FUNCTION_BLOCK fb_auto
VAR_INPUT
END_VAR
VAR_OUTPUT
END_VAR
VAR
	SFCInit: BOOL;
	trn_paramInitDone: BOOL;
	trn_moveToHomeDone: BOOL;
	trn_removeLensDone: BOOL;
	fbi_paramInit: fb_paramInit;
	var_process: INT;
	flg_tranHomeDone: BOOL;
	flg_sampleHomeDone: BOOL;
	flg_trayHomeDone: BOOL;
	flg_chuckHomeDone: BOOL;
	flg_axisHomeDone: BOOL;
	fbi_lensTranport: fb_lensTranport;
	fbi_palletizeing: fb_palletizeing;
	fbi_gm_measurementModule: fb_gm_measurementModule;
	fbi_gm_transport: fb_gm_transport;
	flg_pushHomeDone: BOOL;
	flg_rotaryHomeDone: BOOL;
	trn_measurementSystemHomeDone: BOOL;
	fbi_debuger : fb_debuger;
	fbi_gateLengthList: fb_gateLengthList;
	fbi_dataSampling: fb_dataSampling;
	timer: TON;
	timer2: TON;
	fbi_gm_removeLens: fb_gm_removeLens;
END_VAR

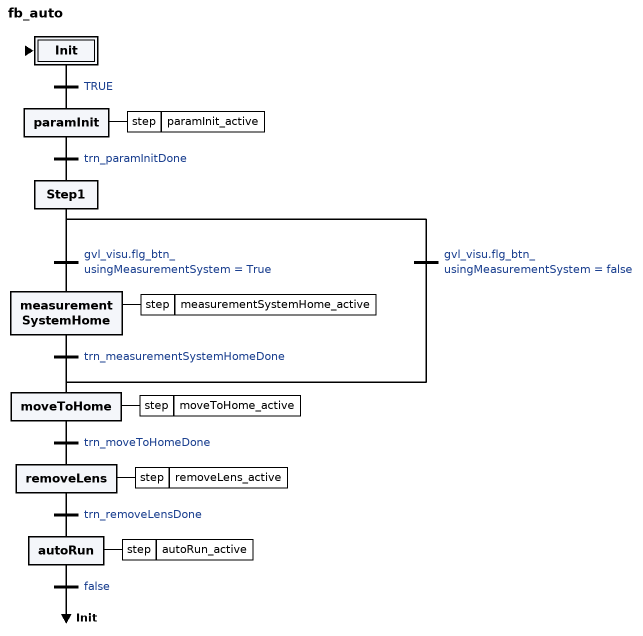
INITIAL_STEP Init:
END_STEP
TRANSITION FROM Init TO paramInit
    := TRUE;
END_TRANSITION
STEP paramInit:
    paramInit_active(N);  // step action
END_STEP
TRANSITION FROM paramInit TO Step1
    := trn_paramInitDone;
END_TRANSITION
STEP Step1:
END_STEP
TRANSITION FROM Step1 TO measurementSystemHome
    := gvl_visu.flg_btn_usingMeasurementSystem = True;
END_TRANSITION
STEP measurementSystemHome:
    measurementSystemHome_active(N);  // step action
END_STEP
TRANSITION FROM measurementSystemHome TO moveToHome
    := trn_measurementSystemHomeDone;
END_TRANSITION
TRANSITION FROM Step1 TO moveToHome
    := gvl_visu.flg_btn_usingMeasurementSystem = false;
END_TRANSITION
STEP moveToHome:
    moveToHome_active(N);  // step action
END_STEP
TRANSITION FROM moveToHome TO removeLens
    := trn_moveToHomeDone;
END_TRANSITION
STEP removeLens:
    removeLens_active(N);  // step action
END_STEP
TRANSITION FROM removeLens TO autoRun
    := trn_removeLensDone;
END_TRANSITION
STEP autoRun:
    autoRun_active(N);  // step action
END_STEP
TRANSITION FROM autoRun TO Init
    := false;
END_TRANSITION

ACTION autoRun_active:
IF autoRun._x AND autoRun.x = FALSE THEN
	THIS^.fbi_lensTranport();
	THIS^.fbi_lensTranport.p_Init := TRUE;
	THIS^.fbi_palletizeing();
	THIS^.fbi_palletizeing.p_Init := TRUE;
	THIS^.fbi_gm_measurementModule.SFCInit := TRUE;
	THIS^.fbi_gm_measurementModule();
	THIS^.fbi_gm_transport();
	THIS^.fbi_gm_transport.p_Init := TRUE;
ELSIF autoRun._x AND autoRun.x THEN
	THIS^.fbi_lensTranport();
	THIS^.fbi_lensTranport.p_Init := FALSE;
	THIS^.fbi_palletizeing();
	THIS^.fbi_palletizeing.p_Init := FALSE;
	IF gvl_visu.flg_btn_usingMeasurementSystem THEN
		THIS^.fbi_gm_measurementModule();
		THIS^.fbi_gm_measurementModule.SFCInit := FALSE;
		THIS^.fbi_gm_transport();
		THIS^.fbi_gm_transport.p_Init := FALSE;
	END_IF
	fbi_dataSampling(
	in_flg_run:= gvl_auto.flg_dataSampling_run, 
	in_var_cavNo:= gvl_auto.buf_cavNo, 
	in_var_pocketNo:= gvl_auto.pocketNo[gvl_auto.buf_cavNo], 
	in_var_gateLength:= gvl_auto.buf_gateLength, 
	in_var_date:= gvl_visu.var_DT, 
	in_flg_nonDefective:= gvl_auto.flg_DataSample_nonDefective, 
	in_flg_defective:= gvl_auto.flg_DataSample_defective, 
	in_flg_sample:= gvl_auto.flg_DataSamle_sample, 
	in_flg_reset:= , 
	ref_dataSet:= gvl_auto.var_DataSet);

	fbi_gateLengthList();
	
	fbi_debuger(
	in_flg_run:= gvl_debug.flg_debug_run, 
	in_flg_start:= gvl_debug.flg_debug_run, 
	in_var_cavQty:= gvl_param.var_productInfo[gvl_param.var_currentProductID].cavQty, 
	out_flg_gateLengthISSuccessed=> gvl_debug.flg_passingMeasurement, 
	out_flg_dummySignal=> , 
	out_flg_lensSetDone=> gvl_debug.out_lensSetDone, 
	out_flg_fiberSens=> gvl_debug.out_fiberSens, 
	out_flg_busy=> gvl_debug.out_busy, 
	out_cav=> gvl_debug.var_cav);
	
END_IF
END_ACTION

ACTION measurementSystemHome_active:
IF measurementSystemHome._x AND measurementSystemHome.x = FALSE THEN
	trn_measurementSystemHomeDone := FALSE;
	gvl_auto.gm_rotaryPowerOn := FALSE;
	var_process := 0;
ELSIF measurementSystemHome._x AND measurementSystemHome.x THEN
	IF gvl_visu.flg_btn_usingMeasurementSystem THEN
		CASE var_process OF
			0://insert parameter
				gvl_solv.fbi_gm_ejector.in_flg_run := FALSE;
				gvl_solv.fbi_gm_chuck.in_flg_run := FALSE;
				gvl_solv.fbi_gm_push.in_flg_run := FALSE;
				gvl_solv.fbi_gm_pickup.in_flg_run := FALSE;
				gvl_solv.fbi_gm_rotary.in_flg_run := FALSE;
				gvl_solv.fbi_gm_stamp.in_flg_run := FALSE;
				gvl_elecylinder.fbi_gm_axisPickUp.in_flg_run := FALSE;
				gvl_elecylinder.fbi_gm_axisTransport.in_flg_run := FALSE;
				gvl_solv.fbi_gm_ejector.in_var_vacMode := eP_ejeVacMode.halt;
				gvl_solv.fbi_gm_chuck.in_var_moveMode := eP_svMoveMode.svA;
				gvl_solv.fbi_gm_push.in_var_moveMode := eP_svMoveMode.svA;
				gvl_solv.fbi_gm_pickup.in_var_moveMode := eP_svMoveMode.svA;
				gvl_solv.fbi_gm_rotary.in_var_moveMode := eP_svMoveMode.svA;
				gvl_solv.fbi_gm_stamp.in_var_moveMode := eP_svMoveMode.svA;
				gvl_elecylinder.fbi_gm_axisPickUp.in_var_moveMode := eP_eleMoveMode.eleA;
				gvl_elecylinder.fbi_gm_axisTransport.in_var_moveMode := eP_eleMoveMode.eleA;
				gvl_axis.ref_r.Position := gvl_param.var_productInfo[gvl_param.var_currentProductID].teachPos.gm_rotary.origin;
				gvl_auto.gm_rotaryPowerOn := TRUE;
				IF gvl_axis.fbi_mc_powerR.Status THEN
					var_process := 1;
				END_IF
			1://first move
				gvl_solv.fbi_gm_ejector.in_flg_run := TRUE;
				gvl_solv.fbi_gm_chuck.in_flg_run := TRUE;
				gvl_solv.fbi_gm_push.in_flg_run := TRUE;
				gvl_elecylinder.fbi_gm_axisPickUp.in_flg_run := TRUE;
				gvl_elecylinder.fbi_gm_axisTransport.in_flg_run := TRUE;
				IF gvl_solv.ref_gm_chuck.in.in_flg_sensA AND
				   gvl_solv.ref_gm_push.in.in_flg_sensA AND
				   gvl_elecylinder.ref_gm_axisPickUp.input.in_flg_sensA AND 
				   gvl_elecylinder.ref_gm_axisTransport.input.in_flg_sensA THEN
				   	gvl_solv.fbi_gm_ejector.in_flg_run := FALSE;
					gvl_solv.fbi_gm_chuck.in_flg_run := FALSE;
					gvl_solv.fbi_gm_push.in_flg_run := FALSE;
					gvl_elecylinder.fbi_gm_axisPickUp .in_flg_run := FALSE;
					gvl_elecylinder.fbi_gm_axisTransport.in_flg_run := FALSE;
					var_process := 2;
				END_IF
			2://second move	
				gvl_axis.ref_r.Execute := TRUE;
				IF gvl_axis.ref_r.Done THEN
					gvl_axis.ref_r.Execute := FALSE;
					var_process := 3;
				END_IF
			3://third move
				gvl_solv.fbi_gm_pickup.in_flg_run := TRUE;
				gvl_solv.fbi_gm_rotary.in_flg_run := TRUE;
				gvl_solv.fbi_gm_stamp.in_flg_run := TRUE;
				IF gvl_solv.ref_gm_pickUp.in.in_flg_sensA AND gvl_solv.ref_gm_rotary.in.in_flg_sensA AND gvl_solv.ref_gm_stamp.in.in_flg_sensA THEN
					var_process := 4;
				END_IF
			4:	
				trn_measurementSystemHomeDone := TRUE;
		END_CASE
		IF gvl_axis.ref_r.Error THEN
			gvl_axis.ref_r.Execute := false;
			var_process := 100;
		END_IF
	ELSE
		trn_measurementSystemHomeDone := TRUE;
	END_IF
END_IF
END_ACTION

ACTION moveToHome_active:
IF moveToHome._x AND moveToHome.x = FALSE THEN
	var_process := 0;
	trn_moveToHomeDone := FALSE;
	gvl_auto.motorPowerOn := FALSE;
ELSIF moveToHome._x AND moveToHome.x THEN
	CASE var_process OF
		0:
			gvl_auto.motorPowerOn := TRUE;
			IF gvl_axis.flg_motorReady THEN
				var_process := 1;
			END_IF
		1://move axisZ
			gvl_axis.ref_z.Position := 0;
			gvl_axis.ref_z.Execute := TRUE;
			IF gvl_axis.ref_z.Done THEN
				gvl_axis.ref_z.Execute := FALSE;
				var_process := 2;
			END_IF
		2://insert parameter
			gvl_solv.fbi_push.in_flg_run := FALSE;
			gvl_elecylinder.fbi_axisTransport.in_var_moveMode := eP_eleMoveMode.eleA;
			gvl_elecylinder.fbi_axisSample.in_var_moveMode := eP_eleMoveMode.eleA;
			gvl_elecylinder.fbi_axisRotary.in_var_moveMode := eP_eleMoveMode.eleA;
			gvl_solv.fbi_chuck.in_var_moveMode := eP_svMoveMode.svA;
			gvl_solv.fbi_push.in_var_moveMode := eP_svMoveMode.svA;
			gvl_elecylinder.fbi_axisTransport.in_flg_run := FALSE;
			gvl_elecylinder.fbi_axisSample.in_flg_run := FALSE;
			gvl_elecylinder.fbi_axisRotary.in_flg_run := FALSE;
			gvl_solv.fbi_chuck.in_flg_run := FALSE;
			gvl_solv.fbi_push.in_flg_run := FALSE;
			gvl_axis.fbi_motionControler.in_flg_start := false;
			gvl_axis.fbi_motionControler.in_var_targetPosX := gvl_param.var_productInfo[gvl_param.var_currentProductID].teachPos.initial.x;
			gvl_axis.fbi_motionControler.in_var_targetPosY := gvl_param.var_productInfo[gvl_param.var_currentProductID].teachPos.initial.y;
			gvl_axis.fbi_motionControler.in_var_targetPosZ := gvl_param.var_productInfo[gvl_param.var_currentProductID].teachPos.initial.z;
			gvl_axis.fbi_motionControler.in_var_direction := eP_motionDirection.XYZ;
			var_process := 3;
		3://moving start
			gvl_elecylinder.fbi_axisTransport.in_flg_run := TRUE;
			gvl_elecylinder.fbi_axisSample.in_flg_run := TRUE;
			gvl_elecylinder.fbi_axisRotary.in_flg_run := TRUE;
			gvl_solv.fbi_chuck.in_flg_run := TRUE;
			gvl_solv.fbi_push.in_flg_run := TRUE;
			gvl_axis.fbi_motionControler.in_flg_start := TRUE;
			IF gvl_elecylinder.fbi_axisTransport.out_flg_Done THEN
				flg_tranHomeDone := TRUE;
			END_IF
			IF gvl_elecylinder.fbi_axisSample.out_flg_Done THEN
				flg_sampleHomeDone := TRUE;
			END_IF
			IF gvl_elecylinder.fbi_axisRotary.out_flg_Done THEN
				flg_rotaryHomeDone := TRUE;
			END_IF
			IF gvl_solv.fbi_chuck.out_flg_Done THEN
				flg_chuckHomeDone := TRUE;
			END_IF
			IF gvl_solv.fbi_push.out_flg_Done THEN
				flg_pushHomeDone := TRUE;
			END_IF
			IF gvl_axis.fbi_motionControler.out_flg_Done THEN
				flg_axisHomeDone := TRUE;
			END_IF 
			IF flg_tranHomeDone AND flg_sampleHomeDone AND flg_chuckHomeDone AND flg_axisHomeDone AND flg_pushHomeDone AND flg_rotaryHomeDone THEN
				var_process := 4;
			END_IF
		4://clear flag
			flg_tranHomeDone := FALSE;
			flg_sampleHomeDone := FALSE;
			flg_chuckHomeDone := FALSE;
			flg_pushHomeDone := FALSE;
			flg_axisHomeDone := FALSE;
			flg_rotaryHomeDone := FALSE;
			gvl_elecylinder.fbi_axisTransport.in_flg_run := FALSE;
			gvl_elecylinder.fbi_axisSample.in_flg_run := FALSE;
			gvl_elecylinder.fbi_axisTrayChange.in_flg_run := FALSE;
			gvl_elecylinder.fbi_axisRotary.in_flg_run := FALSE;
			gvl_solv.fbi_chuck.in_flg_run := FALSE;
			gvl_solv.fbi_push.in_flg_run := FALSE;
			gvl_axis.fbi_motionControler.in_flg_start := FALSE;
			var_process := 5;
		5://check position
			trn_moveToHomeDone := TRUE;			
	END_CASE
END_IF
END_ACTION

PROPERTY p_Init : BOOL
GET
p_Init := THIS^.SFCInit;
END_GET
SET
THIS^.SFCInit := p_Init;
END_SET
END_PROPERTY

ACTION paramInit_active:
IF paramInit._x AND paramInit.x = FALSE THEN
	trn_paramInitDone := FALSE;
	fbi_paramInit.in_flg_run := FALSE;
	THIS^.fbi_lensTranport.p_Init := TRUE;
	THIS^.fbi_lensTranport();
	THIS^.fbi_palletizeing.p_Init := TRUE;
	THIS^.fbi_palletizeing();
	THIS^.fbi_gm_measurementModule.SFCInit := TRUE;
	THIS^.fbi_gm_measurementModule();
	THIS^.fbi_gm_transport();
	THIS^.fbi_gm_transport.p_Init := TRUE;
ELSIF paramInit._x AND paramInit.x THEN
	gvl_auto.gateLengthIsPassed := FALSE;
	gvl_auto.pickUpLnesDone := FALSE;
	gvl_auto.lensVacuumDone := FALSE;
	gvl_auto.requirementToPickUpLens := FALSE;
	gvl_gm.flg_requestPickup := FALSE;
	gvl_gm.flg_lensSetDoneFromGM := FALSE;
	gvl_gm.flg_lensRequest := FALSE;
	gvl_gm.flg_lensPickUpDone := FALSE;
	gvl_debug.flg_debug_run := FALSE;
	gvl_debug.flg_stampDone :=FALSE;
	gvl_debug.flg_stampReady := FALSE;
	gvl_debug.flg_check_quality:= FALSE;
	gvl_debug.flg_to_measurement:= FALSE;
	gvl_debug.flg_to_stocker:= FALSE;
	gvl_visu.flg_btn_vacSensOn := FALSE;
	gvl_visu.flg_btn_gm_motorPower := FALSE;
	gvl_visu.flg_btn_buzzer_silent := FALSE;
	gvl_visu.flg_powerOn := FALSE;
	fbi_paramInit.in_flg_run := TRUE;
	IF fbi_paramInit.out_flg_done THEN
		fbi_paramInit.in_flg_run := FALSE;
		trn_paramInitDone := TRUE;
	END_IF
END_IF

fbi_paramInit(in_flg_run:= , out_flg_done=> );
END_ACTION

ACTION removeLens_active:
IF removeLens._x AND removeLens.x = FALSE THEN
	timer.IN := FALSE;
	timer2.IN := FALSE;
	trn_removeLensDone := FALSE;
	var_process := 0;
ELSIF removeLens._x AND removeLens.x THEN
	CASE var_process OF
		0://insert parameter
			fbi_gm_removeLens.p_Init := TRUE;
			gvl_axis.fbi_motionControler.in_var_targetPosX := gvl_param.var_productInfo[gvl_param.var_currentProductID].teachPos.remove.x;
			gvl_axis.fbi_motionControler.in_var_targetPosY := gvl_param.var_productInfo[gvl_param.var_currentProductID].teachPos.remove.y;
			gvl_axis.fbi_motionControler.in_var_targetPosZ := gvl_param.var_productInfo[gvl_param.var_currentProductID].teachPos.remove.z;
			gvl_axis.fbi_motionControler.in_var_direction := eP_motionDirection.XYZ;
			IF gvl_solv.ref_ejector.input.in_flg_sensVac THEN
				var_process := 1;
			ELSE
				gvl_solv.fbi_ejector.in_var_vacMode := eP_ejeVacMode.break;
				gvl_solv.fbi_ejector.in_flg_run := TRUE;
				var_process := 20;
			END_IF
		1://move start
			gvl_axis.fbi_motionControler.in_flg_start := TRUE;
			IF gvl_axis.fbi_motionControler.out_flg_Done THEN
				var_process := 2;
			END_IF
		2://insert ejector parameter
			gvl_axis.fbi_motionControler.in_flg_start := FALSE;
			gvl_solv.fbi_ejector.in_flg_run := FALSE;
			gvl_solv.fbi_ejector.in_var_vacMode := eP_ejeVacMode.break;
			var_process := 3;
		3://break
			gvl_solv.fbi_ejector.in_flg_run := TRUE;
			IF gvl_solv.fbi_ejector.out_flg_Done THEN
				gvl_solv.fbi_ejector.in_flg_run := FALSE;
				var_process := 4;
			END_IF
		4://insert initial position
			gvl_solv.fbi_ejector.in_flg_run := FALSE;
			gvl_solv.fbi_chuck.in_var_moveMode := eP_svMoveMode.svA;
			gvl_axis.fbi_motionControler.in_var_targetPosX := gvl_param.var_productInfo[gvl_param.var_currentProductID].teachPos.initial.x;
			gvl_axis.fbi_motionControler.in_var_targetPosY := gvl_param.var_productInfo[gvl_param.var_currentProductID].teachPos.initial.y;
			gvl_axis.fbi_motionControler.in_var_targetPosZ := gvl_param.var_productInfo[gvl_param.var_currentProductID].teachPos.initial.z;
			gvl_axis.fbi_motionControler.in_var_direction := eP_motionDirection.ZYX;
			var_process := 5;
		5://move to initial position
			gvl_axis.fbi_motionControler.in_flg_start := TRUE;
			IF gvl_axis.fbi_motionControler.out_flg_Done THEN
				gvl_solv.fbi_gm_push.in_flg_run := FALSE;
				gvl_solv.fbi_gm_chuck.in_flg_run := FALSE;
				IF gvl_io.flg_fiberSens THEN
					var_process := 6;
				ELSE
					var_process := 20;
				END_IF
			END_IF
		6:
			gvl_solv.fbi_chuck.in_var_moveMode := eP_svMoveMode.svB;
			gvl_solv.fbi_push.in_var_moveMode := eP_svMoveMode.svB;
			gvl_elecylinder.fbi_axisTransport.in_var_moveMode := eP_eleMoveMode.eleB;
			gvl_solv.fbi_ejector.in_var_vacMode := eP_ejeVacMode.halt;
			gvl_axis.fbi_motionControler.in_var_targetPosX := gvl_param.var_productInfo[gvl_param.var_currentProductID].teachPos.pickUp.x;
			gvl_axis.fbi_motionControler.in_var_targetPosY := gvl_param.var_productInfo[gvl_param.var_currentProductID].teachPos.pickUp.y;
			gvl_axis.fbi_motionControler.in_var_targetPosZ := gvl_param.var_productInfo[gvl_param.var_currentProductID].teachPos.pickUp.z;
			gvl_axis.fbi_motionControler.in_var_direction := eP_motionDirection.XYZ;
			var_process := 7;
		7:
			gvl_elecylinder.fbi_axisTransport.in_flg_run := TRUE;
			gvl_solv.fbi_ejector.in_flg_run := TRUE;
			gvl_solv.fbi_chuck.in_flg_run := TRUE;
			gvl_solv.fbi_push.in_flg_run := TRUE;
			var_process := 8;
		8:
			IF gvl_io.in_wire_svChuckClose AND gvl_io.in_wire_svPushClose AND gvl_io.in_flg_eleTransportMoving THEN
				gvl_axis.fbi_motionControler.in_flg_start := TRUE;
				gvl_solv.fbi_ejector.in_flg_run := FALSE;
				gvl_elecylinder.fbi_axisTransport.in_flg_run := FALSE;
				gvl_solv.fbi_chuck.in_flg_run := FALSE;
				gvl_solv.fbi_push.in_flg_run := FALSE;
				var_process := 9;
			END_IF
		9:
			IF gvl_axis.fbi_motionControler.out_flg_Done THEN
				gvl_axis.fbi_motionControler.in_flg_start := FALSE;
				gvl_axis.fbi_motionControler.in_var_targetPosX := gvl_param.var_productInfo[gvl_param.var_currentProductID].teachPos.initial.x;
				gvl_axis.fbi_motionControler.in_var_targetPosY := gvl_param.var_productInfo[gvl_param.var_currentProductID].teachPos.initial.y;
				gvl_axis.fbi_motionControler.in_var_targetPosZ := gvl_param.var_productInfo[gvl_param.var_currentProductID].teachPos.initial.z;
				gvl_axis.fbi_motionControler.in_var_direction := eP_motionDirection.ZYX;
				var_process := 10;
			END_IF
		10:
			gvl_axis.fbi_motionControler.in_flg_start := TRUE;
			var_process := 11;
		11:
			IF gvl_axis.fbi_motionControler.out_flg_Done THEN
				gvl_axis.fbi_motionControler.in_flg_start := FALSE;
				gvl_axis.fbi_motionControler.in_var_targetPosX := gvl_param.var_productInfo[gvl_param.var_currentProductID].teachPos.remove.x;
				gvl_axis.fbi_motionControler.in_var_targetPosY := gvl_param.var_productInfo[gvl_param.var_currentProductID].teachPos.remove.y;
				gvl_axis.fbi_motionControler.in_var_targetPosZ := gvl_param.var_productInfo[gvl_param.var_currentProductID].teachPos.remove.z;
				gvl_axis.fbi_motionControler.in_var_direction := eP_motionDirection.XYZ;
				var_process := 12;
			END_IF
		12:
			gvl_axis.fbi_motionControler.in_flg_start := TRUE;
			gvl_solv.fbi_ejector.in_var_vacMode := eP_ejeVacMode.break;
			var_process := 13;
		13:
			IF gvl_axis.fbi_motionControler.out_flg_Done THEN
				gvl_solv.fbi_ejector.in_flg_run := TRUE;
				var_process := 14;	
			END_IF
		14:
			IF gvl_solv.fbi_ejector.out_flg_Done THEN
				gvl_solv.fbi_ejector.in_flg_run := FALSE;
				gvl_axis.fbi_motionControler.in_var_targetPosX := gvl_param.var_productInfo[gvl_param.var_currentProductID].teachPos.initial.x;
				gvl_axis.fbi_motionControler.in_var_targetPosY := gvl_param.var_productInfo[gvl_param.var_currentProductID].teachPos.initial.y;
				gvl_axis.fbi_motionControler.in_var_targetPosZ := gvl_param.var_productInfo[gvl_param.var_currentProductID].teachPos.initial.z;
				gvl_axis.fbi_motionControler.in_var_direction := eP_motionDirection.ZYX;
				var_process := 15;	
			END_IF
		15:
			gvl_axis.fbi_motionControler.in_flg_start := TRUE;
			gvl_solv.fbi_chuck.in_var_moveMode := eP_svMoveMode.svB;
			gvl_solv.fbi_push.in_var_moveMode := eP_svMoveMode.svB;
			gvl_elecylinder.fbi_axisTransport.in_var_moveMode := eP_eleMoveMode.eleB;
			var_process := 16;
		16:
			IF gvl_axis.fbi_motionControler.out_flg_Done THEN
				IF gvl_axis.fbi_motionControler.out_flg_Done THEN
					gvl_elecylinder.fbi_axisTransport.in_flg_run := TRUE;
					gvl_solv.fbi_chuck.in_flg_run := TRUE;
					gvl_solv.fbi_push.in_flg_run := TRUE;
					var_process := 17;
				END_IF
			END_IF
		17:
			IF gvl_io.in_wire_svChuckOpen AND gvl_io.in_wire_svPushOpen AND gvl_io.in_flg_eleTransportOrigin THEN
				gvl_elecylinder.fbi_axisTransport.in_flg_run := FALSE;
				gvl_solv.fbi_chuck.in_flg_run := FALSE;
				gvl_solv.fbi_push.in_flg_run := FALSE;
				var_process := 20;
			END_IF
		20:
			IF NOT gvl_visu.flg_btn_usingMeasurementSystem THEN
				var_process := 50;
			ELSE
				fbi_gm_removeLens.p_Init := TRUE;
				fbi_gm_removeLens.in_flg_run := FALSE;
				var_process := 21;
			END_IF
		21:
			fbi_gm_removeLens.p_Init := FALSE;
			fbi_gm_removeLens.in_flg_run := TRUE;
			var_process := 22;
		22:
			fbi_gm_removeLens.in_flg_run := FALSE;
			IF fbi_gm_removeLens.out_flg_Done THEN
				var_process := 50;
			END_IF
			
		50:
			gvl_solv.fbi_ejector.in_flg_run := FALSE;
			trn_removeLensDone := TRUE;
	END_CASE
	fbi_gm_removeLens(in_flg_run:= , out_flg_Done=> );
	timer(IN:= , PT:= T#0.5S , Q=> , ET=> );
	timer2(IN:= , PT:= T#0.5S , Q=> , ET=> );
END_IF
END_ACTION

END_FUNCTION_BLOCK

(* stored: Version 1.1.0.1, ProductVersion 3.1.4024.11
   POU fb_auto: Id {45b3f956-88f7-486e-97f8-ae993956690a}, SpecialFunc None
   Action autoRun_active: Id {6e20425c-d870-46e8-8c79-c42919ac8af5}
   Action measurementSystemHome_active: Id {1bb8f388-2672-415a-b6ef-d9bf552f8ea9}
   Action moveToHome_active: Id {16d02ed0-296b-4321-886b-30e2802ea8ea}
   Property p_Init: Id {c2d0da88-466b-4d96-8bc5-090a73b1a683}
   Get Get: Id {049645de-0c21-46cb-b025-7b12ce1ac435}
   Set Set: Id {a7055906-8822-44fe-844c-79624dc22269}
   Action paramInit_active: Id {3554c9c6-7cc2-4335-ba5f-a6a21c001791}
   Action removeLens_active: Id {c740f2c1-662e-4a4b-82ef-bf592dd0c6fd} *)
